(* PLC project Unnamed, Unknown Unnamed 1 *)
(* stored: creationDateTime 2020-03-04T10:06:13, modificationDateTime 2020-03-06T12:45:27 *)

FUNCTION_BLOCK principal
  VAR_OUTPUT
    ST1 : BOOL;
    ST2 : BOOL;
    ST3 : BOOL;
    ST4 : BOOL;
    ST5 : BOOL;
    ST6 : BOOL;
    ST7 : BOOL;
    ST8 : BOOL;
    ST9 : BOOL;
    ST10 : BOOL;
    ST11 : BOOL;
    ST16 : BOOL;
    ST17 : BOOL;
    ST18 : BOOL;
  END_VAR
  VAR_INPUT
    M_LAVAGE : BOOL;  (* M0 *)
    M_RINSE : BOOL;  (* M1 *)
    M_HOT_RINSE : BOOL;  (* M2 *)
    M_P_SAVON : BOOL;  (* M3 *)
    M_P_ASSAIN : BOOL;  (* M4 *)
    M_DRAINAGE : BOOL;  (* M5 *)
    M_DELAI_VIDANGE : BOOL;  (* M24 *)
    M_FLOTTE : BOOL;  (* M35 *)
    DEPART : BOOL;  (* I0 *)
    WATER_SAVER : BOOL;  (* I2 *)
    CYCLE_3 : BOOL;  (* I3 *)
    URGENCEZ : BOOL;  (* I4 *)
    BOOSTER_READY : BOOL;  (* I10 *)
    HEATER : BOOL;  (* I11 *)
  END_VAR

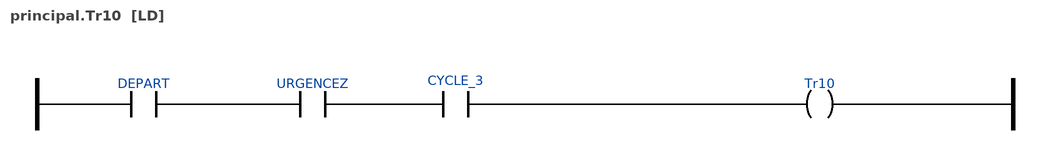
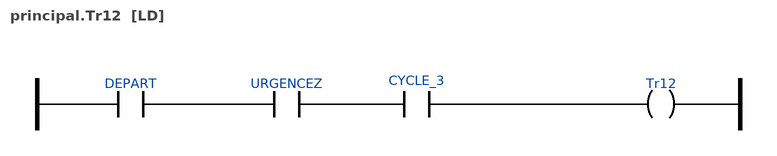
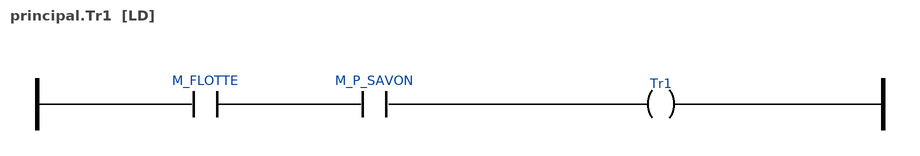
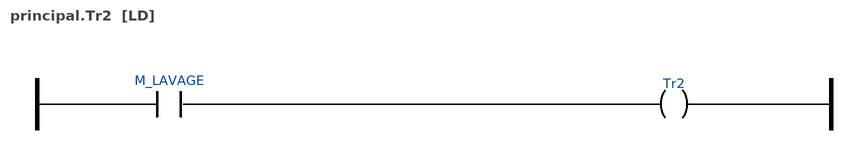
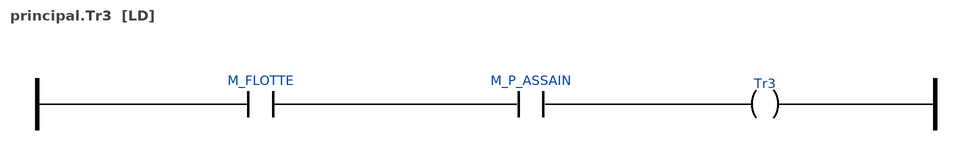
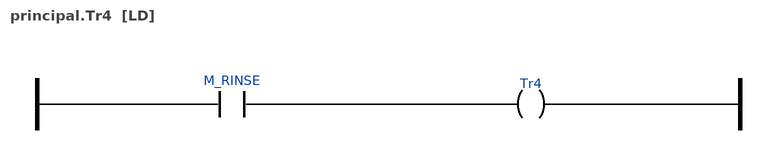
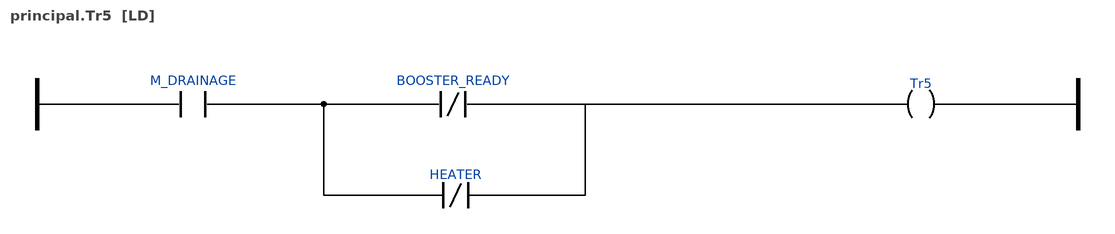
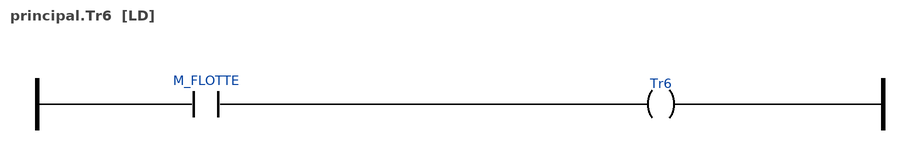
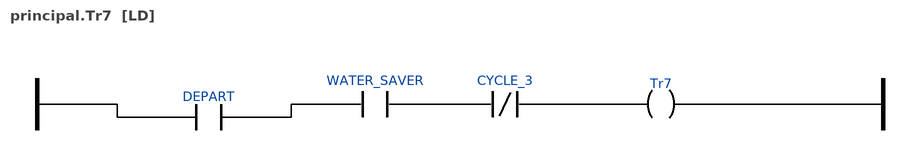
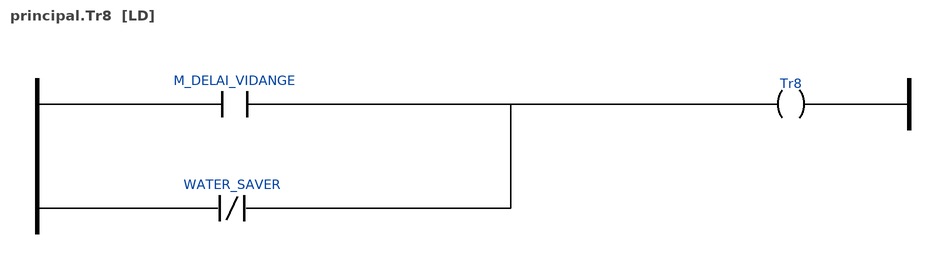
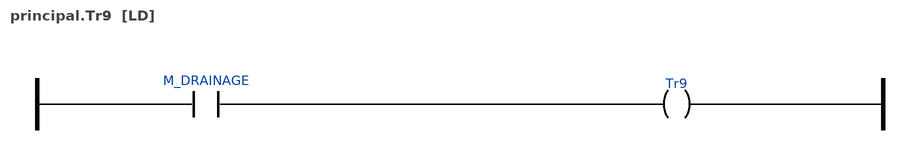
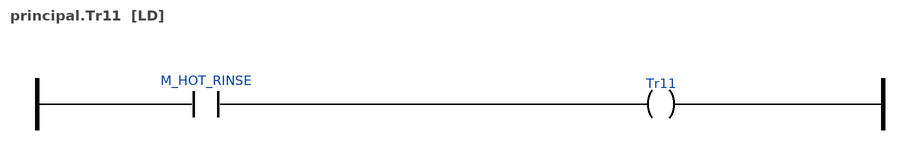
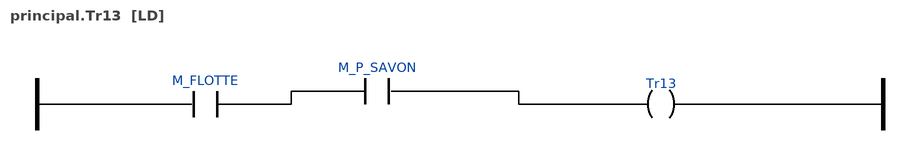
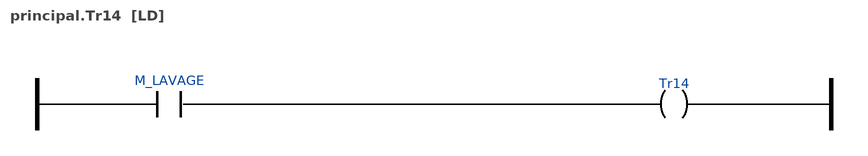
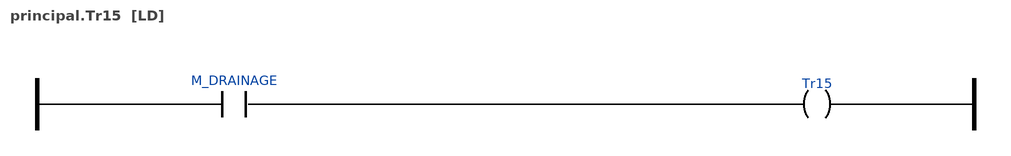
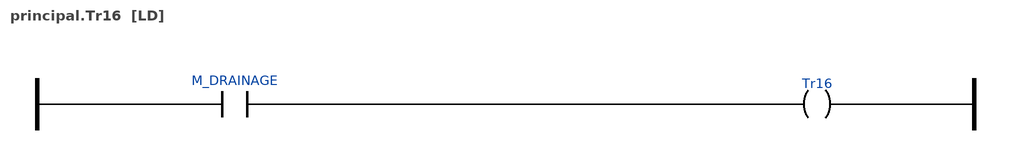
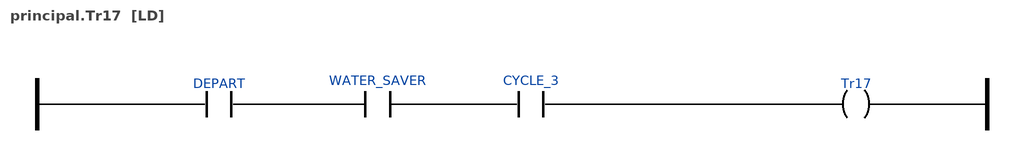
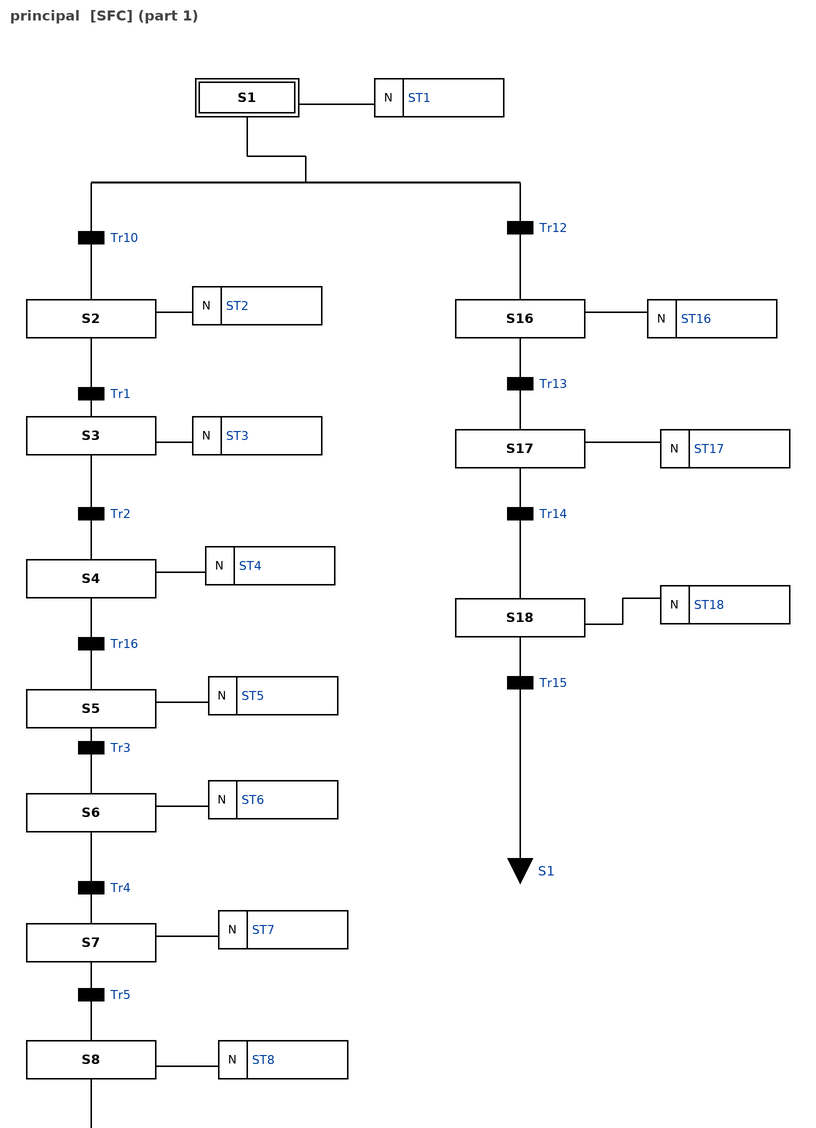
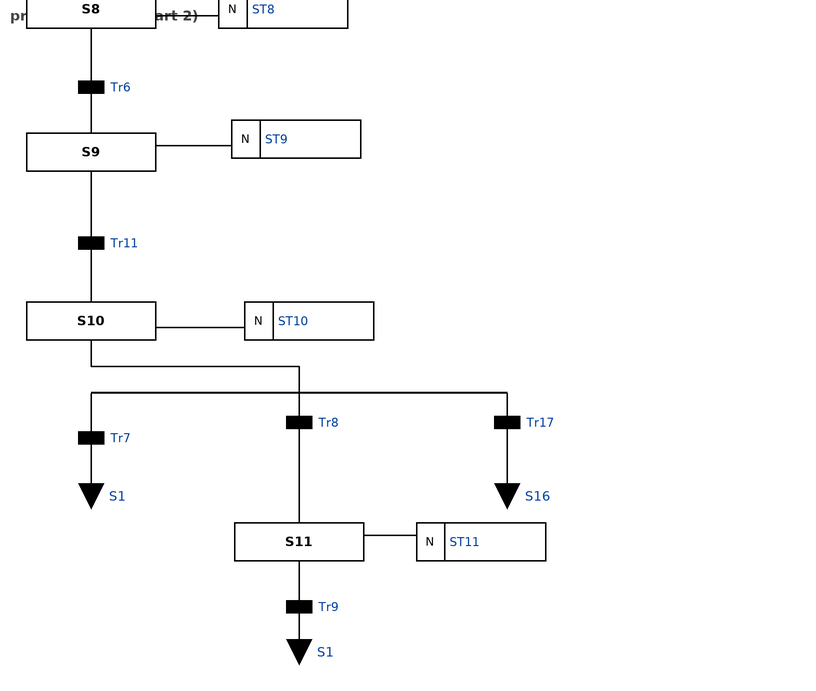
INITIAL_STEP S1:
  ST1(N);
END_STEP
TRANSITION FROM S1 TO S2  (* Tr10 *)
  := DEPART AND URGENCEZ AND CYCLE_3;
END_TRANSITION
TRANSITION FROM S1 TO S16  (* Tr12 *)
  := DEPART AND URGENCEZ AND CYCLE_3;
END_TRANSITION
STEP S2:
  ST2(N);
END_STEP
TRANSITION FROM S2 TO S3  (* Tr1 *)
  := M_FLOTTE AND M_P_SAVON;
END_TRANSITION
STEP S16:
  ST16(N);
END_STEP
TRANSITION FROM S16 TO S17  (* Tr13 *)
  := M_FLOTTE AND M_P_SAVON;
END_TRANSITION
STEP S3:
  ST3(N);
END_STEP
TRANSITION FROM S3 TO S4  (* Tr2 *)
  := M_LAVAGE;
END_TRANSITION
STEP S17:
  ST17(N);
END_STEP
TRANSITION FROM S17 TO S18  (* Tr14 *)
  := M_LAVAGE;
END_TRANSITION
STEP S4:
  ST4(N);
END_STEP
TRANSITION FROM S4 TO S5  (* Tr16 *)
  := M_DRAINAGE;
END_TRANSITION
STEP S18:
  ST18(N);
END_STEP
TRANSITION FROM S18 TO S1  (* Tr15 *)
  := M_DRAINAGE;
END_TRANSITION
STEP S5:
  ST5(N);
END_STEP
TRANSITION FROM S5 TO S6  (* Tr3 *)
  := M_FLOTTE AND M_P_ASSAIN;
END_TRANSITION
STEP S6:
  ST6(N);
END_STEP
TRANSITION FROM S6 TO S7  (* Tr4 *)
  := M_RINSE;
END_TRANSITION
STEP S7:
  ST7(N);
END_STEP
TRANSITION FROM S7 TO S8  (* Tr5 *)
  := M_DRAINAGE AND (NOT BOOSTER_READY OR NOT HEATER);
END_TRANSITION
STEP S8:
  ST8(N);
END_STEP
TRANSITION FROM S8 TO S9  (* Tr6 *)
  := M_FLOTTE;
END_TRANSITION
STEP S9:
  ST9(N);
END_STEP
TRANSITION FROM S9 TO S10  (* Tr11 *)
  := M_HOT_RINSE;
END_TRANSITION
STEP S10:
  ST10(N);
END_STEP
TRANSITION FROM S10 TO S1  (* Tr7 *)
  := DEPART AND WATER_SAVER AND NOT CYCLE_3;
END_TRANSITION
TRANSITION FROM S10 TO S11  (* Tr8 *)
  := M_DELAI_VIDANGE OR NOT WATER_SAVER;
END_TRANSITION
TRANSITION FROM S10 TO S16  (* Tr17 *)
  := DEPART AND WATER_SAVER AND CYCLE_3;
END_TRANSITION
STEP S11:
  ST11(N);
END_STEP
TRANSITION FROM S11 TO S1  (* Tr9 *)
  := M_DRAINAGE;
END_TRANSITION
END_FUNCTION_BLOCK

FUNCTION_BLOCK urgence
  VAR_OUTPUT
    ST12 : BOOL;
    ST13 : BOOL;
    ST14 : BOOL;
    ST15 : BOOL;
  END_VAR
  VAR_INPUT
    DEPART : BOOL;  (* I0 *)
    URGENCES : BOOL;  (* I4 *)
    M_DRAINAGE : BOOL;  (* M5 *)
    M_STEP_1 : BOOL;  (* M6 *)
  END_VAR

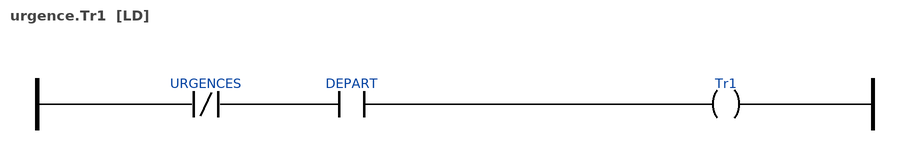
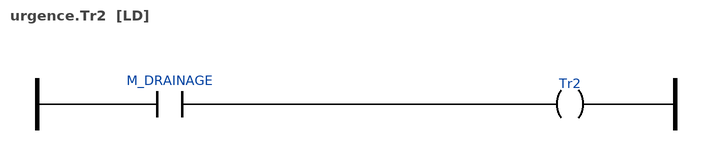
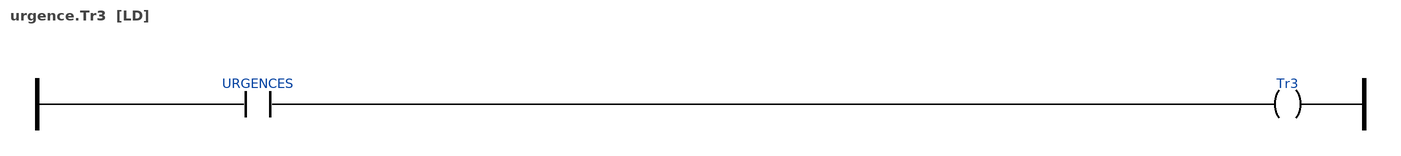
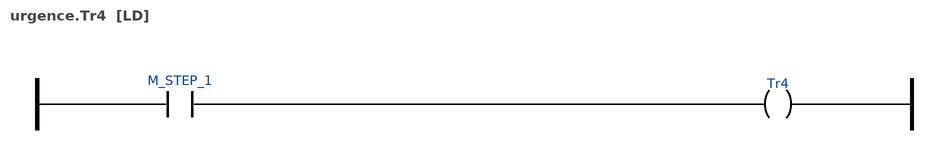
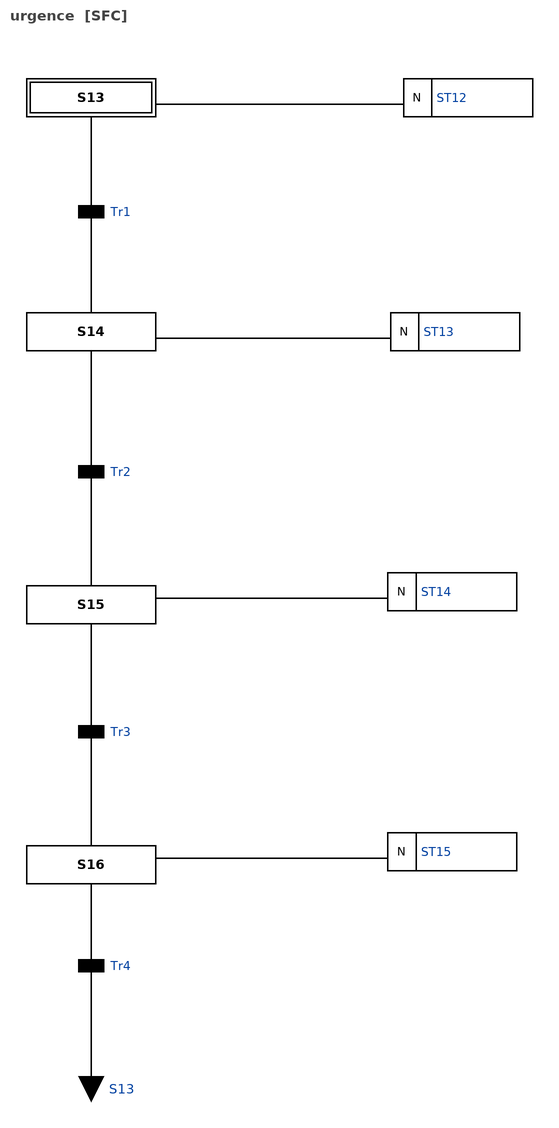
INITIAL_STEP S13:
  ST12(N);
END_STEP
TRANSITION FROM S13 TO S14  (* Tr1 *)
  := NOT URGENCES AND DEPART;
END_TRANSITION
STEP S14:
  ST13(N);
END_STEP
TRANSITION FROM S14 TO S15  (* Tr2 *)
  := M_DRAINAGE;
END_TRANSITION
STEP S15:
  ST14(N);
END_STEP
TRANSITION FROM S15 TO S16  (* Tr3 *)
  := URGENCES;
END_TRANSITION
STEP S16:
  ST15(N);
END_STEP
TRANSITION FROM S16 TO S13  (* Tr4 *)
  := M_STEP_1;
END_TRANSITION
END_FUNCTION_BLOCK

PROGRAM general
  VAR
    TAMPON_CHAUFFAGE : TON;
    T_OVERFLOW : TON;
    T_POMPE_SAVON : TON;
    T_DRAIN : TON;
    T_POMPE_SAVON_3_EXTRA : TON;
    T_POMPE_SANI : TON;
    T_LAVAGE : TON;
    T_PRE_WASH : TON;
    T_DELAI_VIDANGE : TON;
    T_HOT_RINSE : TON;
    T_ASSAIN : TON;
    DELAI_MOTEUR : TON;
    T_BRAS_LAVAGE_1 : TON;
    T_BRAS_LAVAGE_3 : TON;
    T_BRAS_LAVAGE_2 : TON;
    T_BRAS_PRE_LAVAGE_3 : TON;
    T_BRAS_ASSAIN_1 : TON;
    T_BRAS_ASSAIN_2 : TON;
    T_BRAS_ASSAIN_3 : TON;
    T_BRAS_HOT_RINCE_1 : TON;
    T_BRAS_HOT_RINCE_2 : TON;
    T_BRAS_HOT_RINCE_3 : TON;
    T_ALARME_FIN_DE_CYCLE : TON;
    urgence0 : urgence;
    principal0 : principal;
    STEP_1 : BOOL;  (* X0 *)
    STEP_2 : BOOL;  (* X1 *)
    STEP_3 : BOOL;  (* X2 *)
    STEP_4 : BOOL;  (* X3 *)
    STEP_5 : BOOL;  (* X4 *)
    STEP_6 : BOOL;  (* X5 *)
    STEP_7 : BOOL;  (* X6 *)
    STEP_8 : BOOL;  (* X7 *)
    STEP_9 : BOOL;  (* X8 *)
    STEP_10 : BOOL;  (* X9 *)
    STEP_11 : BOOL;  (* X10 *)
    STEP_12 : BOOL;  (* X11 *)
    STEP_13 : BOOL;  (* X12 *)
    STEP_14 : BOOL;  (* X13 *)
    STEP_15 : BOOL;  (* X14 *)
    STEP_16 : BOOL;  (* X15 *)
    STEP_17 : BOOL;  (* X16 *)
    STEP_18 : BOOL;  (* X17 *)
  END_VAR
  VAR
    DEPART AT %IX0.0 : BOOL;  (* I0 *)
    CYCLE_1 AT %IX0.1 : BOOL;  (* I1 *)
    WATER_SAVER AT %IX0.2 : BOOL;  (* I2 *)
    CYCLE_3 AT %IX0.3 : BOOL;  (* I3 *)
    URGENCEL AT %IX0.4 : BOOL;  (* I4 *)
    COUVERT AT %IX0.5 : BOOL;  (* I5 *)
    FLOTTE_BASSIN_BAS AT %IX0.6 : BOOL;  (* I6 *)
    FLOTTE_BOOSTER AT %IX0.7 : BOOL;  (* I7 *)
    FLOTTE_BASSIN_HAUT AT %IX1.0 : BOOL;  (* I8 *)
    SELECTEUR_LO_LEVEL AT %IX1.1 : BOOL;  (* I9 *)
    BOOSTER_READY AT %IX1.2 : BOOL;  (* I10 *)
    HEATER AT %IX1.3 : BOOL;  (* I11 *)
    MOTEUR AT %QX2.0 : BOOL;  (* Q0 *)
    DRAIN AT %QX2.1 : BOOL;  (* Q1 *)
    BUZZER AT %QX2.2 : BOOL;  (* Q2 *)
    CHAUFFAGE AT %QX2.3 : BOOL;  (* Q3 *)
    EAU_BOOSTER AT %QX2.4 : BOOL;  (* Q4 *)
    EAU_FRAICHE AT %QX2.5 : BOOL;  (* Q5 *)
    POMPE_SAVON AT %QX2.6 : BOOL;  (* Q6 *)
    POMPE_ASSAIN AT %QX2.7 : BOOL;  (* Q7 *)
    LUMIERE_VERTE AT %QX3.0 : BOOL;  (* Q8 *)
    LUMIERE_JAUNE AT %QX3.1 : BOOL;  (* Q9 *)
    BRAS_DE_LAVAGE AT %QX3.2 : BOOL;  (* Q10 *)
    unused0 AT %QX3.3 : BOOL;  (* Q11 *)
    unused1 AT %QX3.4 : BOOL;  (* Q12 *)
    unused2 AT %QX3.5 : BOOL;  (* Q13 *)
  END_VAR
  VAR
    M_LAVAGE : BOOL;  (* M0 *)
    M_RINSE : BOOL;  (* M1 *)
    M_HOT_RINSE : BOOL;  (* M2 *)
    M_P_SAVON : BOOL;  (* M3 *)
    M_P_ASSAIN : BOOL;  (* M4 *)
    M_DRAINAGE : BOOL;  (* M5 *)
    M_STEP_1 : BOOL;  (* M6 *)
    M_STEP_2 : BOOL;  (* M7 *)
    M_DRAIN : BOOL;  (* M8 *)
    M_FICTIVE : BOOL;  (* M9 *)
    M_STEP_3 : BOOL;  (* M10 *)
    M_STEP_4 : BOOL;  (* M11 *)
    M_STEP_5 : BOOL;  (* M12 *)
    M_STEP_6 : BOOL;  (* M13 *)
    M_STEP_7 : BOOL;  (* M14 *)
    M_STEP_8 : BOOL;  (* M15 *)
    M_STEP_9 : BOOL;  (* M16 *)
    M_STEP_10 : BOOL;  (* M17 *)
    M_STEP_11 : BOOL;  (* M18 *)
    M_STEP_12 : BOOL;  (* M19 *)
    M_STEP_13 : BOOL;  (* M20 *)
    M_STEP_14 : BOOL;  (* M21 *)
    M_STEP_15 : BOOL;  (* M22 *)
    M_STEP_16 : BOOL;  (* M23 *)
    M_DELAI_VIDANGE : BOOL;  (* M24 *)
    M_DELAI_MOTEUR : BOOL;  (* M25 *)
    M_STEP_17 : BOOL;  (* M26 *)
    M_STEP_18 : BOOL;  (* M27 *)
    M_TAMPON_CHAUFFAGE : BOOL;  (* M28 *)
    M_BRAS : BOOL;  (* M29 *)
    M_BRAS_2 : BOOL;  (* M30 *)
    M_STEP_22 : BOOL;  (* M31 *)
    M_OVERFLOW : BOOL;  (* M32 *)
    M_ALARM_OVERFLOW : BOOL;  (* M33 *)
    M_FIN_DE_CYCLE : BOOL;  (* M34 *)
    M_FLOTTE : BOOL;  (* M35 *)
    M_BRAS_3 : BOOL;  (* M36 *)
    SB_INTERGRAFCET : BOOL;  (* M36 *)
    SB_FIRSTRUN : BOOL;  (* M36 *)
  END_VAR

